PROGRAM OvenExample
VAR
	oven : OvenBasic;
	heatCall : PLCopenCall;
	startHeating : BOOL;
	desiredTemp : REAL;
END_VAR

oven.cyclic();

IF startHeating THEN
	oven.StartHeating(desiredTemp,heatCall);
	startHeating := 0;
END_IF

heatCall();
heatCall.Execute := 0;

IF heatCall.Done THEN
	//do the next thing
END_IF

END_PROGRAM

(* stored: Version 1.1.0.1
   POU OvenExample: Id {b57ab83e-29e5-0abb-0aa3-87f8d2927bf3}, SpecialFunc None *)
